// TwinCAT 3 PLC project SendingMQTT
// ProgramVersion: 3.1.4022.3
// libraries:
//   Tc2_Standard, * (Beckhoff Automation GmbH)
//   Tc2_System, * (Beckhoff Automation GmbH)
//   Tc2_Utilities, * (Beckhoff Automation GmbH)
//   Tc3_IotBase, * (Beckhoff Automation GmbH)
//   Tc3_IotCommunicator, * (Beckhoff Automation GmbH)
//   Tc3_JsonXml, * (Beckhoff Automation GmbH)
//   Tc3_Module, * (Beckhoff Automation GmbH)
// project tree:
//   DUTs/ ST_TemperatureStructure.TcDUT
//   GVLs/ Data_Published.TcGVL, Setup_Parameters.TcGVL
//   / PlcTask.TcTTO
//   POUs/ FB_GenerateData.TcPOU, MAIN_Publisher.TcPOU
// real-time tasks:
//   TASK PlcTask: cycle T#10ms, priority 20, ADS port 350

CONFIGURATION SendingMQTT
    RESOURCE PLC ON TwinCAT3
        TASK PlcTask(INTERVAL := T#10ms, PRIORITY := 20);
        PROGRAM MAIN_Publisher WITH PlcTask : MAIN_Publisher;
    END_RESOURCE
END_CONFIGURATION

// ---- DUTs/ST_TemperatureStructure.TcDUT
TYPE ST_TemperatureStructure :
STRUCT
	fRoomTemperature 		: REAL	:= 21;
	fBathRoomTemperature 	: REAL	:= 18;
	diSomeOtherData 		: DINT	:= 1124;
END_STRUCT
END_TYPE

// ---- GVLs/Data_Published.TcGVL
{attribute 'qualified_only'}
VAR_GLOBAL
	stTempData	: ST_TemperatureStructure;	// this is the data that we will publish to our MQTT topic.

	// String representation of data for MQQT messages
	sJsonFormattedDataString	: STRING(255); //JSON formatted string
    sPlainFormattedDataString	: STRING(255); //plain formatted string 
	
	// Count the messages sent
	uiSent						: UINT;
	
END_VAR

// ---- GVLs/Setup_Parameters.TcGVL
{attribute 'qualified_only'}
VAR_GLOBAL CONSTANT
	sPlainStringTopic	: STRING(255)	:= 'Plain Temperatures';	// this the topic we will publish on for plain string data
	sJsonStringTopic	: STRING(255)	:= 'JSON Temperatures';		// this the topic we will publish on for JSON formatted string data
	sBrokerAddress		: STRING(255)	:= 'test.mosquitto.org';	// this is the address of the MQTT broker we are using
	uiBrokerPort 		: UINT			:= 1883;					// the TCP port for the MQQT broker
	tUpdateTime			: TIME			:= T#5S;					// the update time
END_VAR

// ---- POUs/MAIN_Publisher.TcPOU
PROGRAM MAIN_Publisher
VAR
	fbMqttClient				: FB_IotMqttClient; 	// MQTT client.       
    fbSendUpdateIntervalTimer 	: TON := (PT:=Setup_Parameters.tUpdateTime);	// Interval timer for broadcasting( we send updated data when this timer runs out) .
	
	fbJsonWriter 	: FB_JsonSaxWriter;			// function block for writing JSON formatted string 
	fbJsonDataType 	: FB_JsonReadWriteDataType;	// function block for getting JSON formatted string representation of a STRUCT
	fbGetSystemTime	: GETSYSTEMTIME;
	fbNoisyData		: FB_GenerateData;
		
END_VAR

// We setup out MQTT client, only happens on the first run of the PLC code
fbGetSystemTime();
IF _TaskInfo[GETCURTASKINDEXEX()].FirstCycle THEN    
    fbMqttClient.sHostName      := Setup_Parameters.sBrokerAddress;
    fbMqttClient.nHostPort      := Setup_Parameters.uiBrokerPort;
    fbMqttClient.sTopicPrefix   := '';     
	fbMqttClient.sClientId 		:= CONCAT('Publishing_PLC_',DWORD_TO_STRING(fbGetSystemTime.timeLoDW));	// generate and set a psuedorandom client ID 
END_IF

// Generate some noisy data
fbNoisyData(bRun:= TRUE,pDataStructure:=ADR(Data_Published.stTempData));

// We run the MQTT client every cycle
fbMqttClient.Execute(TRUE);

IF fbMqttClient.bConnected THEN	// chekc that the MQTT client is connected to the broker
    fbSendUpdateIntervalTimer(IN:=TRUE);		// run our send update timer  
    IF fbSendUpdateIntervalTimer.Q THEN			// if the timer has expired (its time to send an update) 
        fbSendUpdateIntervalTimer(IN:=FALSE);  	// reset our send update timer
     
		// Generate out plain formatted string from the data structure
        Data_Published.sPlainFormattedDataString := CONCAT(CONCAT(CONCAT('*Room temperature:',REAL_TO_STRING(Data_Published.stTempData.fRoomTemperature)),CONCAT('*Bathroom temperature:',REAL_TO_STRING(Data_Published.stTempData.fBathRoomTemperature))),CONCAT('*Some other data:',DINT_TO_STRING(Data_Published.stTempData.diSomeOtherData)));
		
		// Publish our plain formatted string message using our MQTT client
        fbMqttClient.Publish(	sTopic		:= Setup_Parameters.sPlainStringTopic, 
        						pPayload	:= ADR(Data_Published.sPlainFormattedDataString), 
								nPayloadSize:= LEN2(ADR(Data_Published.sPlainFormattedDataString))+1, 
            					eQoS		:= TcIotMqttQos.AtMostOnceDelivery, 
								bRetain		:= FALSE,
								bQueue		:= FALSE);
			
			
		// Generate a JSON formatted string representing the data structure
		fbJsonWriter.ResetDocument();
		fbJsonDataType.AddJsonValueFromSymbol(fbJsonWriter, 'ST_TemperatureStructure', SIZEOF(Data_Published.stTempData), ADR(Data_Published.stTempData));
		Data_Published.sJsonFormattedDataString := fbJsonWriter.GetDocument();	// we get the JSON string that the fbJsonDataType FB has generated for us
			
		// Publish our JSON formatted string message using our MQTT client
		fbMqttClient.Publish(	sTopic		:= Setup_Parameters.sJsonStringTopic, 
								pPayload	:= ADR(Data_Published.sJsonFormattedDataString), 
								nPayloadSize:= LEN2(ADR(Data_Published.sJsonFormattedDataString))+1, 
								eQoS		:= TcIotMqttQos.AtMostOnceDelivery, 
								bRetain		:= FALSE,
								bQueue		:= FALSE);

		Data_Published.uiSent	:= Data_Published.uiSent + 1;	// count the messages sent  
    END_IF // Update timer elapsed
END_IF // Client connected

END_PROGRAM

// ---- POUs/FB_GenerateData.TcPOU
FUNCTION_BLOCK FB_GenerateData
VAR_INPUT
	bRun			: BOOL;
	pDataStructure	: POINTER TO ST_TemperatureStructure;
END_VAR
VAR_OUTPUT
END_VAR
VAR
	fbGetSystemTime	: GETSYSTEMTIME;
END_VAR

fbGetSystemTime();
IF(bRun)THEN
	IF(pDataStructure <>0)THEN
		pDataStructure^.fRoomTemperature		:= 21 + pDataStructure^.fRoomTemperature * SIN(fbGetSystemTime.timeLoDW);
		pDataStructure^.fBathRoomTemperature	:= 18 + pDataStructure^.fBathRoomTemperature * COS(fbGetSystemTime.timeLoDW);
		pDataStructure^.diSomeOtherData			:= pDataStructure^.diSomeOtherData + (DWORD_TO_DINT(fbGetSystemTime.timeLoDW));
	END_IF
END_IF

END_FUNCTION_BLOCK
